(* IEC 61131-3 sources: SIMATIC-AX-Tutorial/src, 3 files *)

(* ---- function.st ---- *)
FUNCTION Power : LINT
    VAR_INPUT
        x : LINT;
    END_VAR
Power := x * x;
END_FUNCTION

(* ---- configuration.st ---- *)
CONFIGURATION MyConfiguration
    TASK Main(Interval := T#500ms, Priority := 1);
    PROGRAM P1 WITH Main: MyProgram;

        VAR_GLOBAL
            toggle : BOOL;                                   //defines a variable of type bool with name toggle
            output_signal AT %Q0.1 : BOOL;
            input_signal AT %IW2 : WORD;                  //defines a output signal of type bool with name output_signal at PLC adress %Q0.1
            count_value : LINT;                              //defines a variable of type LINT with name count_value
            power_value : LINT;                              //defines a variable of type LINT with name power_value
          END_VAR
END_CONFIGURATION

(* ---- program.st ---- *)
USING System.Counters;

PROGRAM MyProgram
   VAR_EXTERNAL
      toggle : BOOL;
      output_signal : BOOL;
      count_value : LINT;
      power_value : LINT;
   END_VAR
   VAR
      count : CounterUp := (presetValue := 5);
   END_VAR
   toggle := NOT toggle;
   count(up := toggle);
   output_signal := count.presetReached;
   count_value := count.value;
   count.reset := count_value >= 15;
   power_value := Power(count_value);
END_PROGRAM
